// TwinCAT 3 PLC project Fraktal_Modules
// Title: Fraktal_Modules
// Company: fraktal-automation
// Author: fraktal-automation
// ProjectVersion: 0.1.0.2
// Description: Reusable Fraktal module library: cylinder CMs, clamp EM, simulation models, and configured device presets. Reason bands 10100s/11000s per Core 8.8.
// ProgramVersion: 3.1.4024.0
// libraries:
//   Tc2_Standard, * (Beckhoff Automation GmbH)
//   Tc2_System, * (Beckhoff Automation GmbH)
//   Tc2_Utilities, * (Beckhoff Automation GmbH)
//   Tc3_Module, * (Beckhoff Automation GmbH)
//   Fraktal_Core, 0.1.0.3 (fraktal-automation)
// project tree:
//   DUTs/ E_ConfigurableCylinderCommand.TcDUT, E_ClampCommand.TcDUT, E_CylinderCommand.TcDUT, E_CylinderPosition.TcDUT, E_PowerGroupCommand.TcDUT, ST_TwoHandHal.TcDUT, ST_TwoHandParCfg.TcDUT, ST_TwoHandParCmd.TcDUT, ST_TwoHandOutCmd.TcDUT, ST_TwoHandOutImm.TcDUT, ST_PneumaticPressParCfg.TcDUT, ST_PneumaticPressParCmd.TcDUT, ST_PneumaticPressOutCmd.TcDUT, ST_PneumaticPressOutImm.TcDUT, ST_PowerGroupHal.TcDUT, ST_PowerGroupParCfg.TcDUT, ST_PowerGroupParCmd.TcDUT, ST_PowerGroupOutCmd.TcDUT, ST_PowerGroupOutImm.TcDUT, ST_ConfigurableCylinderParCfg.TcDUT, ST_ConfigurableCylinderParCmd.TcDUT, ST_ConfigurableCylinderOutCmd.TcDUT, ST_ConfigurableCylinderOutImm.TcDUT, ST_ConfigurableCylinderHal.TcDUT, ST_ClampParCfg.TcDUT, ST_ClampStationParCfg.TcDUT, ST_ClampStationParCmd.TcDUT, ST_ClampStationOutCmd.TcDUT, ST_ClampStationOutImm.TcDUT, ST_ClampParCmd.TcDUT, ST_ClampOutCmd.TcDUT, ST_ClampOutImm.TcDUT, ST_CylinderHal.TcDUT, ST_CylinderParCfg.TcDUT, ST_CylinderParCmd.TcDUT, ST_CylinderOutCmd.TcDUT, ST_CylinderOutImm.TcDUT, ST_CylinderIoIdentity.TcDUT, ST_DigitalInputHal.TcDUT, ST_DigitalInputOutImm.TcDUT, ST_AirPressureHal.TcDUT, ST_AirPressureOutImm.TcDUT
//   / FB_ConfigurableCylinderCM.TcPOU, FB_ConfigurableCylinderSim.TcPOU, FB_ClampEM.TcPOU, FB_ClampStationUnit.TcPOU, FB_CylinderCM.TcPOU, FB_DigitalInputCM.TcPOU, FB_AirPressureMonitorCM.TcPOU, FB_CylinderSim.TcPOU, FB_Iv3VisionCM.TcPOU, FB_Matrix220CM.TcPOU, FB_PowerGroupCM.TcPOU, FB_TwoHandStartCM.TcPOU
//   Params/ PL_ModuleReasons.TcGVL

// ---- DUTs/E_ConfigurableCylinderCommand.TcDUT
{attribute 'qualified_only'}
TYPE E_ConfigurableCylinderCommand : (NONE := 0, TO_HOME := 1, TO_WORK := 2) DINT;
END_TYPE

// ---- DUTs/E_ClampCommand.TcDUT
{attribute 'qualified_only'}
TYPE E_ClampCommand : (NONE := 0, CLAMP := 1, UNCLAMP := 2) DINT;
END_TYPE

// ---- DUTs/E_CylinderCommand.TcDUT
{attribute 'qualified_only'}
TYPE E_CylinderCommand : (NONE := 0, EXTEND := 1, RETRACT := 2) DINT;
END_TYPE

// ---- DUTs/E_CylinderPosition.TcDUT
// Basic cylinder position (Home = retracted rest, Work = extended active).
{attribute 'qualified_only'}
TYPE E_CylinderPosition : (UNKNOWN := 0, HOME := 1, WORK := 2, MID := 3) DINT;
END_TYPE

// ---- DUTs/E_PowerGroupCommand.TcDUT
{attribute 'qualified_only'}
TYPE E_PowerGroupCommand : (NONE := 0, POWER_ON := 1, POWER_OFF := 2) DINT;
END_TYPE

// ---- DUTs/ST_TwoHandHal.TcDUT
// Raw button status plus the certified safety application's evaluated result.
// SafeActive is never calculated by the standard PLC in a real machine.
TYPE ST_TwoHandHal :
STRUCT
    LeftPressed     : BOOL;
    RightPressed    : BOOL;
    SafeActive      : BOOL;
    FieldbusHealthy : BOOL;
END_STRUCT
END_TYPE

// ---- DUTs/ST_TwoHandParCfg.TcDUT
TYPE ST_TwoHandParCfg :
STRUCT
    SchemaVersion : UINT := 1;
    RequireReleaseBetweenCycles : BOOL := TRUE;
END_STRUCT
END_TYPE

// ---- DUTs/ST_TwoHandParCmd.TcDUT
TYPE ST_TwoHandParCmd :
STRUCT
    Reserved : BOOL;
END_STRUCT
END_TYPE

// ---- DUTs/ST_TwoHandOutCmd.TcDUT
TYPE ST_TwoHandOutCmd :
STRUCT
    StartAccepted : BOOL;
END_STRUCT
END_TYPE

// ---- DUTs/ST_TwoHandOutImm.TcDUT
TYPE ST_TwoHandOutImm :
STRUCT
    LeftPressed     : BOOL;
    RightPressed    : BOOL;
    SafeActive      : BOOL;
    Armed           : BOOL;
    StartPulse      : BOOL;
    FieldbusHealthy : BOOL;
    Diagnostic      : ST_Diagnostic;
END_STRUCT
END_TYPE

// ---- DUTs/ST_PneumaticPressParCfg.TcDUT
// Core §3.8 ParCfg (SchemaVersion first; adding a member = schema change).
// v2 adds the §8.11 performance references: per-model ideal cycle (OEE
// Performance denominator, §8.5.1) and the WORK-time degradation baseline
// (§8.11.4(d); 0 = watch off).
TYPE ST_PneumaticPressParCfg :
STRUCT
    SchemaVersion       : UINT := 2;
    PressSettleTime     : TIME := T#500MS;
    TransferSettleTime  : TIME := T#100MS;
    RequireTwoHandStart : BOOL := TRUE;
    IdealCycleMs        : UDINT := 0;    // §8.5.1 — 0 = Performance not computed
    BaselineWorkMs      : UDINT := 0;    // §8.11.4(d) — 0 = degradation watch off
END_STRUCT
END_TYPE

// ---- DUTs/ST_PneumaticPressParCmd.TcDUT
TYPE ST_PneumaticPressParCmd :
STRUCT
    Reserved : BOOL;
END_STRUCT
END_TYPE

// ---- DUTs/ST_PneumaticPressOutCmd.TcDUT
TYPE ST_PneumaticPressOutCmd :
STRUCT
    CycleCompleted : BOOL;
    Homed          : BOOL;
    ChangeoverCompleted : BOOL;
END_STRUCT
END_TYPE

// ---- DUTs/ST_PneumaticPressOutImm.TcDUT
TYPE ST_PneumaticPressOutImm :
STRUCT
    PressRetracted  : BOOL;
    DoorOpen        : BOOL;
    DoorClosed      : BOOL;
    SlideInside     : BOOL;
    SlideOutside    : BOOL;
    TwoHandArmed    : BOOL;
    TwoHandActive   : BOOL;
    PartPresent     : BOOL;
    AirPressureOk   : BOOL;
    ReadyForLoad    : BOOL;
    ActiveSettleTime: TIME;
    Diagnostic      : ST_Diagnostic;
END_STRUCT
END_TYPE

// ---- DUTs/ST_PowerGroupHal.TcDUT
TYPE ST_PowerGroupHal :
STRUCT
    EnableRequestOut : BOOL; // untrusted functional request; safety system remains authoritative
    PowerFeedback    : BOOL;
    SafetyPermit     : BOOL; // read-only alias from certified safety application
    FieldbusHealthy  : BOOL;
END_STRUCT
END_TYPE

// ---- DUTs/ST_PowerGroupParCfg.TcDUT
TYPE ST_PowerGroupParCfg :
STRUCT
    SchemaVersion        : UINT := 1;
    Kind                 : E_PowerGroupKind;
    RequiredForControl   : BOOL := TRUE;
    FieldbusLossReaction : E_FieldbusLossReaction := E_FieldbusLossReaction.CONTROL_OFF;
    FeedbackTimeout      : TIME := T#2S;
END_STRUCT
END_TYPE

// ---- DUTs/ST_PowerGroupParCmd.TcDUT
TYPE ST_PowerGroupParCmd :
STRUCT
    SchemaVersion : UINT := 1;
END_STRUCT
END_TYPE

// ---- DUTs/ST_PowerGroupOutCmd.TcDUT
TYPE ST_PowerGroupOutCmd :
STRUCT
    PowerOn : BOOL;
END_STRUCT
END_TYPE

// ---- DUTs/ST_PowerGroupOutImm.TcDUT
TYPE ST_PowerGroupOutImm :
STRUCT
    Status     : ST_PowerGroupStatus;
    Diagnostic : ST_Diagnostic;
END_STRUCT
END_TYPE

// ---- DUTs/ST_ConfigurableCylinderParCfg.TcDUT
// Core §3.8 ParCfg (SchemaVersion first). Basic cylinder with optional, possibly
// REDUNDANT, position sensors. Values live in the module that needs them (§3.8a).
TYPE ST_ConfigurableCylinderParCfg :
STRUCT
    SchemaVersion     : UINT := 1;

    // --- optional & redundant sensors ---
    // count of sensors wired for each position: 0 = sensorless (time-based),
    // 1 = single, 2 = duplex (AND-combined), up to PL_Fraktal.MAX_POS_SENSORS.
    HomeSensorCount   : INT := 1;
    WorkSensorCount   : INT := 1;

    // --- timing ---
    MoveTimeout       : TIME := T#5S;    // max movement time (default 5 s)
    SettleTime        : TIME := T#30MS;  // debounce before a move is declared done
    TravelTime        : TIME := T#1S;    // sensorless travel assumption (< MoveTimeout)
    DiscrepancyTime   : TIME := T#500MS; // how long redundant sensors may disagree before fault

    // --- behaviour ---
    SingleActing      : BOOL := FALSE;   // TRUE: only ToWorkOut driven; spring return home
    SafePosOnAbort    : E_CylinderPosition := E_CylinderPosition.HOME;
    DeenergizeOnAbort : BOOL := TRUE;
END_STRUCT
END_TYPE

// ---- DUTs/ST_ConfigurableCylinderParCmd.TcDUT
TYPE ST_ConfigurableCylinderParCmd :
STRUCT
    Reserved : BOOL;
END_STRUCT
END_TYPE

// ---- DUTs/ST_ConfigurableCylinderOutCmd.TcDUT
TYPE ST_ConfigurableCylinderOutCmd :
STRUCT
    ReachedPosition : E_CylinderPosition;
END_STRUCT
END_TYPE

// ---- DUTs/ST_ConfigurableCylinderOutImm.TcDUT
TYPE ST_ConfigurableCylinderOutImm :
STRUCT
    Position   : E_CylinderPosition;
    AtHome     : BOOL;
    AtWork     : BOOL;
    Diagnostic : ST_Diagnostic;
END_STRUCT
END_TYPE

// ---- DUTs/ST_ConfigurableCylinderHal.TcDUT
// Basic cylinder HAL with REDUNDANT position sensors (safety cylinders).
// Each position has an array of sensors; only the first N (ParCfg.*SensorCount) are
// used. N = 0 -> sensorless (time-based completion). 'Arrived' = ALL present
// sensors TRUE (AND); a persistent split faults (discrepancy monitoring, §3.6.
TYPE ST_ConfigurableCylinderHal :
STRUCT
    ToWorkOut : BOOL;   // solenoid: drive to work (extend)
    ToHomeOut : BOOL;   // solenoid: drive to home (retract); single-acting leaves FALSE
    HomeFb    : ARRAY[1..PL_Fraktal.MAX_POS_SENSORS] OF BOOL;   // redundant home sensors
    WorkFb    : ARRAY[1..PL_Fraktal.MAX_POS_SENSORS] OF BOOL;   // redundant work sensors
END_STRUCT
END_TYPE

// ---- DUTs/ST_ClampParCfg.TcDUT
TYPE ST_ClampParCfg :
STRUCT
    SchemaVersion : UINT := 1;
    SettleTime    : TIME := T#150MS;
END_STRUCT
END_TYPE

// ---- DUTs/ST_ClampStationParCfg.TcDUT
TYPE ST_ClampStationParCfg :
STRUCT
    SchemaVersion : UINT := 1;
END_STRUCT
END_TYPE

// ---- DUTs/ST_ClampStationParCmd.TcDUT
TYPE ST_ClampStationParCmd :
STRUCT
    Reserved : BOOL;
END_STRUCT
END_TYPE

// ---- DUTs/ST_ClampStationOutCmd.TcDUT
TYPE ST_ClampStationOutCmd :
STRUCT
    CycleCompleted : BOOL;
END_STRUCT
END_TYPE

// ---- DUTs/ST_ClampStationOutImm.TcDUT
TYPE ST_ClampStationOutImm :
STRUCT
    Clamped   : BOOL;
    Unclamped : BOOL;
    Diagnostic: ST_Diagnostic;
END_STRUCT
END_TYPE

// ---- DUTs/ST_ClampParCmd.TcDUT
TYPE ST_ClampParCmd :
STRUCT
    Reserved : BOOL;
END_STRUCT
END_TYPE

// ---- DUTs/ST_ClampOutCmd.TcDUT
TYPE ST_ClampOutCmd :
STRUCT
    Confirmed : BOOL;
END_STRUCT
END_TYPE

// ---- DUTs/ST_ClampOutImm.TcDUT
TYPE ST_ClampOutImm :
STRUCT
    Clamped    : BOOL;
    Unclamped  : BOOL;
    Diagnostic : ST_Diagnostic;
END_STRUCT
END_TYPE

// ---- DUTs/ST_CylinderHal.TcDUT
// Annex B — cylinder HAL: 2 outputs, 2 position sensors
TYPE ST_CylinderHal :
STRUCT
    ExtendOut, RetractOut   : BOOL;
    ExtendedFb, RetractedFb : BOOL;
END_STRUCT
END_TYPE

// ---- DUTs/ST_CylinderParCfg.TcDUT
// Core §3.8: SchemaVersion FIRST, initialized to the expected version
TYPE ST_CylinderParCfg :
STRUCT
    SchemaVersion : UINT := 1;
    MoveTimeout   : TIME := T#2S;
END_STRUCT
END_TYPE

// ---- DUTs/ST_CylinderParCmd.TcDUT
TYPE ST_CylinderParCmd :
STRUCT
    Reserved : BOOL;
END_STRUCT
END_TYPE

// ---- DUTs/ST_CylinderOutCmd.TcDUT
TYPE ST_CylinderOutCmd :
STRUCT
    Reached : BOOL;
END_STRUCT
END_TYPE

// ---- DUTs/ST_CylinderOutImm.TcDUT
TYPE ST_CylinderOutImm :
STRUCT
    Extended   : BOOL;
    Retracted  : BOOL;
    ExtendedSensorTag : STRING(80);
    RetractedSensorTag: STRING(80);
    ExtendOutputTag   : STRING(80);
    RetractOutputTag  : STRING(80);
    Diagnostic : ST_Diagnostic;
END_STRUCT
END_TYPE

// ---- DUTs/ST_CylinderIoIdentity.TcDUT
// Physical identity injection for the four semantic I/O roles of a cylinder.
// The reusable CM never knows terminal models, channel numbers or project tags.
TYPE ST_CylinderIoIdentity :
STRUCT
    ExtendedSensor : ST_IoPointIdentity;
    RetractedSensor : ST_IoPointIdentity;
    ExtendOutput : ST_IoPointIdentity;
    RetractOutput : ST_IoPointIdentity;
    ExtendedTimeoutKey : STRING(255);
    RetractedTimeoutKey : STRING(255);
    BothSensorsKey : STRING(255);
END_STRUCT
END_TYPE

// ---- DUTs/ST_DigitalInputHal.TcDUT
TYPE ST_DigitalInputHal :
STRUCT
    Value : BOOL;
    Quality : BOOL := TRUE;
END_STRUCT
END_TYPE

// ---- DUTs/ST_DigitalInputOutImm.TcDUT
TYPE ST_DigitalInputOutImm :
STRUCT
    Value : BOOL;
    Quality : BOOL;
    IoTag : STRING(80);
    Diagnostic : ST_Diagnostic;
END_STRUCT
END_TYPE

// ---- DUTs/ST_AirPressureHal.TcDUT
TYPE ST_AirPressureHal :
STRUCT
    LowPressure : BOOL;
    OperatingPressure : BOOL;
    Quality : BOOL := TRUE;
END_STRUCT
END_TYPE

// ---- DUTs/ST_AirPressureOutImm.TcDUT
TYPE ST_AirPressureOutImm :
STRUCT
    LowPressure : BOOL;
    OperatingPressure : BOOL;
    PressureOk : BOOL;
    Contradictory : BOOL;
    Quality : BOOL;
    LowSensorTag : STRING(80);
    OperatingSensorTag : STRING(80);
    Diagnostic : ST_Diagnostic;
END_STRUCT
END_TYPE

// ---- Params/PL_ModuleReasons.TcGVL
{attribute 'qualified_only'}
// Core §8.8 band constants (band-extensibility rule): cylinder CM 10100-10199,
// clamp EM 11000-11999 — registered in the Core §8.8 registry.
VAR_GLOBAL CONSTANT
    CYL_NOT_EXTENDED    : DINT := 10101;
    CYL_NOT_RETRACTED   : DINT := 10102;
    CYL_BOTH_SENSORS    : DINT := 10103;
    CLAMP_NOT_CONFIRMED : DINT := 11001;
    // basic cylinder 10200-10299
    CYL_HOME_NOT_REACHED : DINT := 10111;   // timeout moving to home
    CYL_WORK_NOT_REACHED : DINT := 10112;   // timeout moving to work
    CYL_POS_IMPLAUSIBLE  : DINT := 10113;   // home AND work sensor confirmed at once (implausible)
    CYL_SENSOR_LOST      : DINT := 10114;   // confirmed position sensor dropped while holding
    CYL_DISCREPANCY      : DINT := 10116;   // redundant sensors for one position disagree > DiscrepancyTime
    CYL_CFG_INVALID      : DINT := 10115;   // TravelTime >= MoveTimeout, or no sensor+no travel
    // power-group CM 10500-10599
    POWER_ENABLE_WITHHELD : DINT := 10501;
    POWER_FEEDBACK_TIMEOUT: DINT := 10502;
    // air-pressure monitor CM 10600-10699
    AIR_SWITCH_CONFLICT    : DINT := 10601;
END_VAR

// ---- FB_ConfigurableCylinderCM.TcPOU
// Production-grade basic pneumatic cylinder Control Module (Core §2.2 base) with
// OPTIONAL and REDUNDANT position sensors (safety cylinders). Per position: 0..N
// sensors; 0 = sensorless (time-based). 'Arrived' = ALL present sensors TRUE (AND,
// safest); a persistent split of redundant sensors faults (discrepancy monitoring).
// The type is ONLY its device logic; lifecycle/timing/first-out/abort are inherited.
{attribute 'OPC.UA.DA' := '1'}
FUNCTION_BLOCK FB_ConfigurableCylinderCM EXTENDS FB_ControlModuleBase
VAR_INPUT
    Command : E_ConfigurableCylinderCommand;
    ParCfg : ST_ConfigurableCylinderParCfg;
    ParCmd : ST_ConfigurableCylinderParCmd;
END_VAR
VAR_OUTPUT
    OutCmd : ST_ConfigurableCylinderOutCmd;
    OutImm : ST_ConfigurableCylinderOutImm;
    Intlk  : FB_PermIntlk;
END_VAR
VAR
    _hal     : REFERENCE TO ST_ConfigurableCylinderHal;
    _recipe  : I_RecipeProvider;
    _tMove   : TON;
    _tSettle : TON;
    _tDiscH  : TON;                             // home discrepancy timer
    _tDiscW  : TON;                             // work discrepancy timer
    _cfgOk   : BOOL;
    _force   : BOOL;                            // SIM-only interlock force (§5.7)
    _parCfgStaged : ST_ConfigurableCylinderParCfg;
    _recipePrepared : BOOL;
END_VAR

Cyclic();

METHOD Setup : BOOL
VAR_INPUT
    Name   : STRING(80);
    HalRef : REFERENCE TO ST_ConfigurableCylinderHal;
    Recipe : I_RecipeProvider;
END_VAR
VAR
    InitialModel : ST_ModelId;
END_VAR
_M_SetName(Name);
_M_SetPresentation(DisplayNameKey := 'std.moduleType.configurableCylinder.name', DescriptionKey := 'std.moduleType.configurableCylinder.description');
_M_PublishCommand(Value := TO_DINT(E_ConfigurableCylinderCommand.TO_HOME), Label := 'std.command.toHome');   // §7.6.1 catalog
_M_PublishCommand(Value := TO_DINT(E_ConfigurableCylinderCommand.TO_WORK), Label := 'std.command.toWork');
_hal REF= HalRef;                                        // [TC3] TC3 §3.11
_recipe := Recipe;
Intlk.Define(Index := 1, Description := 'project.interlock.areaSafe', Reason := E_Reason.INTERLOCK_DROPPED, Bypassable := FALSE);
Setup := PrepareRecipe(Model := InitialModel);
IF Setup THEN CommitRecipe(); END_IF
END_METHOD

METHOD PrepareRecipe : BOOL
VAR_INPUT
    Model : ST_ModelId;
END_VAR
_parCfgStaged := ParCfg;
IF _recipe <> 0 THEN
    IF NOT _recipe.Load(ModelCode := Model.ModelCode, RecipeKey := 'ConfigurableCylinderCM', pParCfg := ADR(_parCfgStaged), Size := SIZEOF(_parCfgStaged)) THEN
        _M_Fault(E_Reason.RECIPE_INVALID, 'std.error.recipeSchemaInvalid');
        PrepareRecipe := FALSE;
        RETURN;
    END_IF
END_IF
// counts within [0..MAX]; sensorless direction needs a usable travel time
_cfgOk := (_parCfgStaged.HomeSensorCount >= 0) AND (_parCfgStaged.HomeSensorCount <= PL_Fraktal.MAX_POS_SENSORS)
      AND (_parCfgStaged.WorkSensorCount >= 0) AND (_parCfgStaged.WorkSensorCount <= PL_Fraktal.MAX_POS_SENSORS)
      AND (_parCfgStaged.TravelTime < _parCfgStaged.MoveTimeout)
      AND ((_parCfgStaged.HomeSensorCount > 0) OR (_parCfgStaged.TravelTime > T#0S))
      AND ((_parCfgStaged.WorkSensorCount > 0) OR (_parCfgStaged.TravelTime > T#0S));
IF NOT _cfgOk THEN
    _M_FaultN(PL_ModuleReasons.CYL_CFG_INVALID, 'std.error.cylinderConfigurationInvalid');
    PrepareRecipe := FALSE;
    RETURN;
END_IF
_recipePrepared := TRUE;
PrepareRecipe := TRUE;
END_METHOD

METHOD CommitRecipe
IF _recipePrepared THEN ParCfg := _parCfgStaged; END_IF
_recipePrepared := FALSE;
END_METHOD

METHOD AbortRecipe
_recipePrepared := FALSE;
END_METHOD

// TRUE iff EVERY wired sensor for the position reads TRUE (AND-combine, safest).
// Count = 0 -> not sensor-decided (caller uses the time path).
METHOD PROTECTED _M_PosArrived : BOOL
VAR_INPUT
    Work : BOOL;    // TRUE = work position, FALSE = home
END_VAR
VAR
    i, n : INT;
    all  : BOOL;
END_VAR
n := SEL(Work, ParCfg.HomeSensorCount, ParCfg.WorkSensorCount);
IF n <= 0 THEN
    _M_PosArrived := FALSE;      // no sensors: caller must use the time-based path
    RETURN;
END_IF
all := TRUE;
FOR i := 1 TO n DO
    IF Work THEN
        IF NOT _hal.WorkFb[i] THEN all := FALSE; END_IF
    ELSE
        IF NOT _hal.HomeFb[i] THEN all := FALSE; END_IF
    END_IF
END_FOR
_M_PosArrived := all;
END_METHOD

// TRUE iff the position's redundant sensors DISAGREE (at least one TRUE and at
// least one FALSE) — the discrepancy condition. Single/zero sensor => never split.
METHOD PROTECTED _M_PosSplit : BOOL
VAR_INPUT
    Work : BOOL;
END_VAR
VAR
    i, n : INT;
    anyT, anyF : BOOL;
END_VAR
n := SEL(Work, ParCfg.HomeSensorCount, ParCfg.WorkSensorCount);
IF n < 2 THEN
    _M_PosSplit := FALSE;
    RETURN;
END_IF
FOR i := 1 TO n DO
    IF Work THEN
        IF _hal.WorkFb[i] THEN anyT := TRUE; ELSE anyF := TRUE; END_IF
    ELSE
        IF _hal.HomeFb[i] THEN anyT := TRUE; ELSE anyF := TRUE; END_IF
    END_IF
END_FOR
_M_PosSplit := anyT AND anyF;
END_METHOD

// live position resolve + discrepancy monitoring (both positions, every scan)
METHOD PROTECTED OnCyclic : DINT
OnCyclic := SUPER^.OnCyclic();
Intlk.Cond[1] := NOT _force;
Intlk();
IF NOT __ISVALIDREF(_hal) THEN
    RETURN;
END_IF
OutImm.AtHome := (ParCfg.HomeSensorCount > 0) AND _M_PosArrived(Work := FALSE);
OutImm.AtWork := (ParCfg.WorkSensorCount > 0) AND _M_PosArrived(Work := TRUE);

// discrepancy monitoring — a persistent split of redundant sensors is a fault
_tDiscH(IN := _M_PosSplit(Work := FALSE), PT := ParCfg.DiscrepancyTime);
_tDiscW(IN := _M_PosSplit(Work := TRUE),  PT := ParCfg.DiscrepancyTime);
IF (_tDiscH.Q OR _tDiscW.Q) AND (_exec <> E_ExecState.ERROR) THEN
    _M_FaultN(PL_ModuleReasons.CYL_DISCREPANCY, 'std.error.cylinderSensorDiscrepancy');
END_IF

// resolve position (AtHome/AtWork already AND-combined)
IF OutImm.AtHome AND OutImm.AtWork THEN
    OutImm.Position := E_CylinderPosition.UNKNOWN;
ELSIF OutImm.AtHome THEN OutImm.Position := E_CylinderPosition.HOME;
ELSIF OutImm.AtWork THEN OutImm.Position := E_CylinderPosition.WORK;
ELSIF (ParCfg.HomeSensorCount > 0) OR (ParCfg.WorkSensorCount > 0) THEN OutImm.Position := E_CylinderPosition.MID;
END_IF
OutImm.Diagnostic := Status.Diagnostic;

// both-positions-active plausibility while idle
IF (_exec = E_ExecState.READY) AND OutImm.AtHome AND OutImm.AtWork THEN
    _M_FaultN(PL_ModuleReasons.CYL_POS_IMPLAUSIBLE, 'std.error.cylinderPositionImplausible');
END_IF
END_METHOD

// §3.14.2 — fail-safe abort
METHOD PROTECTED OnAbort : DINT
OnAbort := SUPER^.OnAbort();
IF NOT __ISVALIDREF(_hal) THEN
    RETURN;
END_IF
IF ParCfg.DeenergizeOnAbort THEN
    _hal.ToWorkOut := FALSE;
    _hal.ToHomeOut := FALSE;
ELSIF ParCfg.SafePosOnAbort = E_CylinderPosition.WORK THEN
    _hal.ToWorkOut := TRUE;  _hal.ToHomeOut := FALSE;
ELSE
    _hal.ToWorkOut := FALSE; _hal.ToHomeOut := NOT ParCfg.SingleActing;
END_IF
END_METHOD

// §5.7 SIM-only
METHOD SimForceInterlock : BOOL
VAR_INPUT
    Ok : BOOL;
END_VAR
_force := NOT Ok;
SimForceInterlock := TRUE;
END_METHOD

// drive -> await (all-sensors-agree, or time when sensorless) -> settle -> done
METHOD PROTECTED _M_Dispatch
VAR
    toWork  : BOOL;
    n       : INT;
    arrived : BOOL;
    d       : ST_Diagnostic;
END_VAR
IF _manualReq THEN
    _manualReq := FALSE;                        // §7.6.1: apply the manual command value
    Command := _manualCmd;                      // routed THROUGH dispatch — interlocks still apply
END_IF
IF (Command <> E_ConfigurableCylinderCommand.TO_HOME) AND (Command <> E_ConfigurableCylinderCommand.TO_WORK) THEN
    _M_Fault(E_Reason.UNSUPPORTED_COMMAND, 'std.error.unsupportedCylinderCommand');
    RETURN;
END_IF
IF Command = E_ConfigurableCylinderCommand.TO_WORK THEN
    _M_TagCommand(Id := 2, Label := 'std.command.toWork');
    toWork := TRUE;
ELSE
    _M_TagCommand(Id := 1, Label := 'std.command.toHome');
    toWork := FALSE;
END_IF
IF NOT Intlk.AllOk THEN
    _hal.ToWorkOut := FALSE;
    _hal.ToHomeOut := FALSE;
    d := Intlk.Diagnostic;
    d.SourcePath := _name;
    _M_FaultDiag(d);
    RETURN;
END_IF
n := SEL(toWork, ParCfg.HomeSensorCount, ParCfg.WorkSensorCount);   // sensors on the TARGET position
CASE _step OF
    10:
        OutCmd.ReachedPosition := E_CylinderPosition.UNKNOWN;
        _hal.ToWorkOut := toWork;
        _hal.ToHomeOut := (NOT toWork) AND (NOT ParCfg.SingleActing);
        _tMove(IN := FALSE);
        _tSettle(IN := FALSE);
        _step := 20;
    20:  // await arrival
        _tMove(IN := TRUE, PT := ParCfg.MoveTimeout);
        IF n > 0 THEN
            arrived := _M_PosArrived(Work := toWork);        // ALL sensors agree
        ELSE
            _tSettle(IN := TRUE, PT := ParCfg.TravelTime);      // sensorless -> travel time
            arrived := _tSettle.Q;
        END_IF
        IF arrived THEN
            _tSettle(IN := FALSE);
            _step := 30;
        ELSIF _tMove.Q THEN
            _tMove(IN := FALSE);
            _M_FaultN(SEL(toWork, PL_ModuleReasons.CYL_HOME_NOT_REACHED, PL_ModuleReasons.CYL_WORK_NOT_REACHED),
                      SEL(toWork, 'std.error.cylinderHomeTimeout', 'std.error.cylinderWorkTimeout'));
        END_IF
    30:  // settle/debounce; re-confirm all sensors still agree
        _tSettle(IN := TRUE, PT := ParCfg.SettleTime);
        IF n <= 0 THEN
            OutCmd.ReachedPosition := SEL(toWork, E_CylinderPosition.HOME, E_CylinderPosition.WORK);
            _M_Complete();
        ELSIF _M_PosArrived(Work := toWork) THEN
            IF _tSettle.Q THEN
                OutCmd.ReachedPosition := SEL(toWork, E_CylinderPosition.HOME, E_CylinderPosition.WORK);
                _M_Complete();
            END_IF
        ELSE
            _tSettle(IN := FALSE);
            _step := 20;                                     // lost agreement; keep waiting in MoveTimeout
        END_IF
ELSE
    _M_Fault(E_Reason.STEP_STALLED, 'std.error.undefinedStep');
END_CASE
END_METHOD

PROPERTY AtPos : E_CylinderPosition
GET
AtPos := OutImm.Position;
END_GET
END_PROPERTY

METHOD PROTECTED _M_PublishStatus
SUPER^._M_PublishStatus();
OutImm.Diagnostic := Status.Diagnostic;
END_METHOD

END_FUNCTION_BLOCK

// ---- FB_ConfigurableCylinderSim.TcPOU
// §5.7 sim plant for FB_ConfigurableCylinderCM with redundant sensors: after a travel time
// it sets all HomeFb[1..HomeN] / WorkFb[1..WorkN] together. StuckWork[i]/StuckHome[i]
// pin a sensor OFF so a test can inject a discrepancy.
FUNCTION_BLOCK FB_ConfigurableCylinderSim
VAR_INPUT
    Travel : TIME := T#100MS;
    HomeN  : INT := 1;
    WorkN  : INT := 1;
    StuckHome : ARRAY[1..PL_Fraktal.MAX_POS_SENSORS] OF BOOL;   // TRUE = pin this sensor OFF
    StuckWork : ARRAY[1..PL_Fraktal.MAX_POS_SENSORS] OF BOOL;
END_VAR
VAR
    _hal : REFERENCE TO ST_ConfigurableCylinderHal;
    _tW, _tH : TON;
    i : INT;
END_VAR

IF NOT __ISVALIDREF(_hal) THEN
    RETURN;
END_IF
_tW(IN := _hal.ToWorkOut, PT := Travel);
IF _tW.Q THEN
    FOR i := 1 TO WorkN DO _hal.WorkFb[i] := NOT StuckWork[i]; END_FOR
    FOR i := 1 TO HomeN DO _hal.HomeFb[i] := FALSE; END_FOR
END_IF
_tH(IN := _hal.ToHomeOut OR (NOT _hal.ToWorkOut AND NOT _hal.ToHomeOut), PT := Travel);
IF _tH.Q THEN
    FOR i := 1 TO HomeN DO _hal.HomeFb[i] := NOT StuckHome[i]; END_FOR
    FOR i := 1 TO WorkN DO _hal.WorkFb[i] := FALSE; END_FOR
END_IF

METHOD Setup : BOOL
VAR_INPUT
    HalRef : REFERENCE TO ST_ConfigurableCylinderHal;
    TravelTime : TIME;
    Home : INT;
    Work : INT;
END_VAR
VAR
    j : INT;
END_VAR
_hal REF= HalRef;
Travel := TravelTime;
HomeN := Home;
WorkN := Work;
FOR j := 1 TO HomeN DO _hal.HomeFb[j] := TRUE; END_FOR   // start at home, all agree
Setup := TRUE;
END_METHOD

END_FUNCTION_BLOCK

// ---- FB_ClampEM.TcPOU
// Annex B on the EM base: orchestration only, no device logic (§3.5); rollup §8.2.
{attribute 'OPC.UA.DA' := '1'}
FUNCTION_BLOCK FB_ClampEM EXTENDS FB_EquipmentModuleBase
VAR_INPUT
    Command : E_ClampCommand;
    ParCfg : ST_ClampParCfg;
    ParCmd : ST_ClampParCmd;
END_VAR
VAR_OUTPUT
    CylA, CylB : FB_CylinderCM;
    OutCmd : ST_ClampOutCmd;
    OutImm : ST_ClampOutImm;
END_VAR
VAR
    _recipe : I_RecipeProvider;
    _tSettle : TON;
    _parCfgStaged : ST_ClampParCfg;
    _recipePrepared : BOOL;
END_VAR

Cyclic();

METHOD PROTECTED OnCyclic : DINT
OnCyclic := SUPER^.OnCyclic();
_M_TickChildren();                       // children stay live (Annex B §B.3)
OutImm.Diagnostic := Status.Diagnostic;
END_METHOD

METHOD PrepareRecipe : BOOL
VAR_INPUT
    Model : ST_ModelId;
END_VAR
IF _recipe = 0 THEN
    _parCfgStaged := ParCfg;
    _recipePrepared := TRUE;
ELSIF _recipe.Load(ModelCode := Model.ModelCode, RecipeKey := 'ClampEM', pParCfg := ADR(_parCfgStaged), Size := SIZEOF(_parCfgStaged)) THEN
    _recipePrepared := TRUE;
ELSE
    _M_Fault(E_Reason.RECIPE_INVALID, 'std.error.recipeSchemaInvalid');
    _recipePrepared := FALSE;
    PrepareRecipe := FALSE;
    RETURN;
END_IF
PrepareRecipe := SUPER^.PrepareRecipe(Model := Model);
IF NOT PrepareRecipe THEN _recipePrepared := FALSE; END_IF
END_METHOD

METHOD CommitRecipe
SUPER^.CommitRecipe();
IF _recipePrepared THEN ParCfg := _parCfgStaged; END_IF
_recipePrepared := FALSE;
END_METHOD

METHOD AbortRecipe
SUPER^.AbortRecipe();
_recipePrepared := FALSE;
END_METHOD

METHOD Setup : BOOL
VAR_INPUT
    Name : STRING(80);
    HalA : REFERENCE TO ST_CylinderHal;
    HalB : REFERENCE TO ST_CylinderHal;
    Recipe : I_RecipeProvider;
END_VAR
VAR
    InitialModel : ST_ModelId;
END_VAR
_M_SetName(Name);
_M_SetPresentation(DisplayNameKey := 'std.moduleType.clamp.name', DescriptionKey := 'std.moduleType.clamp.description');
_recipe := Recipe;
CylA.Setup(Name := CONCAT(Name, '.CylA'), HalRef := HalA, Recipe := Recipe);
CylB.Setup(Name := CONCAT(Name, '.CylB'), HalRef := HalB, Recipe := Recipe);
_M_Register(CylA);
_M_Register(CylB);
_M_PublishCommand(Value := TO_DINT(E_ClampCommand.CLAMP), Label := 'std.command.clamp');
_M_PublishCommand(Value := TO_DINT(E_ClampCommand.UNCLAMP), Label := 'std.command.unclamp');
Setup := PrepareRecipe(Model := InitialModel);
IF Setup THEN CommitRecipe(); END_IF
END_METHOD

METHOD PROTECTED _M_Dispatch
VAR
    dir : E_CylinderCommand;
    ext : BOOL;
END_VAR
IF _manualReq THEN
    _manualReq := FALSE;
    IF (_manualCmd = TO_DINT(E_ClampCommand.CLAMP)) OR (_manualCmd = TO_DINT(E_ClampCommand.UNCLAMP)) THEN
        Command := _manualCmd;
    ELSE
        _M_Fault(E_Reason.UNSUPPORTED_COMMAND, 'std.error.unsupportedClampCommand');
        RETURN;
    END_IF
END_IF
IF (Command <> E_ClampCommand.CLAMP) AND (Command <> E_ClampCommand.UNCLAMP) THEN
    _M_Fault(E_Reason.UNSUPPORTED_COMMAND, 'std.error.unsupportedClampCommand');
    RETURN;
END_IF
ext := (Command = E_ClampCommand.CLAMP);
dir := SEL(ext, E_CylinderCommand.RETRACT, E_CylinderCommand.EXTEND);
IF ext THEN
    _M_TagCommand(Id := 1, Label := 'std.command.clamp');
ELSE
    _M_TagCommand(Id := 2, Label := 'std.command.unclamp');
END_IF
CASE _step OF
    10:  // command both cylinders in parallel (Annex B)
        OutCmd.Confirmed := FALSE;
        CylA.Abort := FALSE;
        CylB.Abort := FALSE;
        CylA.Command := dir;
        CylB.Command := dir;
        CylA.Execute := TRUE;
        CylB.Execute := TRUE;
        _tSettle(IN := FALSE);
        _step := 20;
    20:  // join on both Done — or roll up the first child Error (§8.2)
        IF CylA.Error OR CylB.Error THEN
            _M_RollupFault();
            CylA.Abort := TRUE;                    // stop the partner safely
            CylB.Abort := TRUE;
            CylA.Execute := FALSE;
            CylB.Execute := FALSE;
        ELSIF CylA.Done AND CylB.Done THEN
            CylA.Execute := FALSE;
            CylB.Execute := FALSE;
            _step := 30;
        END_IF
    30:  // settle, then confirm both feedbacks held (EM-level check, Annex B)
        _tSettle(IN := TRUE, PT := ParCfg.SettleTime);
        IF _tSettle.Q THEN
            _tSettle(IN := FALSE);
            IF (ext AND CylA.OutImm.Extended AND CylB.OutImm.Extended)
            OR ((NOT ext) AND CylA.OutImm.Retracted AND CylB.OutImm.Retracted) THEN
                OutImm.Clamped   := ext;
                OutImm.Unclamped := NOT ext;
                OutCmd.Confirmed := TRUE;
                _M_Complete();
            ELSE
                _M_FaultN(PL_ModuleReasons.CLAMP_NOT_CONFIRMED, 'project.error.clampNotConfirmedAfterSettle');
            END_IF
        END_IF
ELSE
    _M_Fault(E_Reason.STEP_STALLED, 'std.error.undefinedStep');
END_CASE
END_METHOD

METHOD PROTECTED _M_PublishStatus
SUPER^._M_PublishStatus();
OutImm.Diagnostic := Status.Diagnostic;
END_METHOD

END_FUNCTION_BLOCK

// ---- FB_CylinderCM.TcPOU
// Annex A/B pattern on the base class: the type is ONLY its device logic.
{attribute 'OPC.UA.DA' := '1'}
FUNCTION_BLOCK FB_CylinderCM EXTENDS FB_ControlModuleBase
VAR_INPUT
    Command : E_CylinderCommand;
    ParCfg : ST_CylinderParCfg;
    ParCmd : ST_CylinderParCmd;
END_VAR
VAR_OUTPUT
    OutCmd : ST_CylinderOutCmd;
    OutImm : ST_CylinderOutImm;
    Intlk  : FB_PermIntlk;
END_VAR
VAR
    _hal    : REFERENCE TO ST_CylinderHal;
    _recipe : I_RecipeProvider;
    _tMove  : TON;
    _force  : BOOL;                     // SIM hook — wrap in {IF defined (SIM_HOOKS)} for release (§5.7)
    _parCfgStaged : ST_CylinderParCfg;
    _recipePrepared : BOOL;
    _directionPermitsConfigured : BOOL;
    _extendPermit, _retractPermit : BOOL := TRUE;
    _extendPermitKey, _retractPermitKey : STRING(255);
    _extendedSensorTag, _retractedSensorTag : STRING(80);
    _extendedSensorAddress, _retractedSensorAddress : STRING(80);
    _extendOutputTag, _retractOutputTag : STRING(80);
    _extendedTimeoutKey, _retractedTimeoutKey, _bothSensorsKey : STRING(255);
    _bothSensorTags, _bothSensorAddresses : STRING(80);
END_VAR

Cyclic();

METHOD PROTECTED OnCyclic : DINT
OnCyclic := SUPER^.OnCyclic();
Intlk.Cond[1] := NOT _force;            // real application: area-safe/air-ok signals (LD/ST, §5.5)
IF NOT _directionPermitsConfigured OR (Command = E_CylinderCommand.NONE) THEN
    Intlk.Cond[2] := TRUE;
ELSIF Command = E_CylinderCommand.EXTEND THEN
    Intlk.Cond[2] := _extendPermit;
ELSIF Command = E_CylinderCommand.RETRACT THEN
    Intlk.Cond[2] := _retractPermit;
ELSE
    Intlk.Cond[2] := FALSE;
END_IF
Intlk();
IF __ISVALIDREF(_hal) THEN              // defensive (§5.6) [TC3]
    OutImm.Extended  := _hal.ExtendedFb;
    OutImm.Retracted := _hal.RetractedFb;
END_IF
OutImm.ExtendedSensorTag := _extendedSensorTag;
OutImm.RetractedSensorTag := _retractedSensorTag;
OutImm.ExtendOutputTag := _extendOutputTag;
OutImm.RetractOutputTag := _retractOutputTag;
OutImm.Diagnostic := Status.Diagnostic;
END_METHOD

// Schematic identity is application configuration, not device behavior.
// Diagnostics keep SourcePath as this module and add the exact failed channel.
METHOD ConfigureIoIdentity
VAR_INPUT
    Identity : ST_CylinderIoIdentity;
END_VAR
_extendedSensorTag := Identity.ExtendedSensor.Tag;
_extendedSensorAddress := Identity.ExtendedSensor.Address;
_retractedSensorTag := Identity.RetractedSensor.Tag;
_retractedSensorAddress := Identity.RetractedSensor.Address;
_extendOutputTag := Identity.ExtendOutput.Tag;
_retractOutputTag := Identity.RetractOutput.Tag;
_extendedTimeoutKey := Identity.ExtendedTimeoutKey;
_retractedTimeoutKey := Identity.RetractedTimeoutKey;
_bothSensorsKey := Identity.BothSensorsKey;
_bothSensorTags := CONCAT(Identity.ExtendedSensor.Tag, CONCAT(' / ', Identity.RetractedSensor.Tag));
_bothSensorAddresses := CONCAT(Identity.ExtendedSensor.Address, CONCAT(' / ', Identity.RetractedSensor.Address));
END_METHOD

// Functional stop used by an owning sequence on abort/interlock loss.
// This is not a certified stop; the safety system remains authoritative.
METHOD WithdrawOutputs
IF __ISVALIDREF(_hal) THEN
    _hal.ExtendOut := FALSE;
    _hal.RetractOut := FALSE;
END_IF
END_METHOD

METHOD PROTECTED OnAbort : DINT
OnAbort := SUPER^.OnAbort();            // base first (§3.14.2)
IF __ISVALIDREF(_hal) THEN
    _hal.ExtendOut := FALSE;
    _hal.RetractOut := FALSE;
END_IF
END_METHOD

METHOD PrepareRecipe : BOOL
VAR_INPUT
    Model : ST_ModelId;
END_VAR
IF _recipe = 0 THEN
    _parCfgStaged := ParCfg;
    _recipePrepared := TRUE;
    PrepareRecipe := TRUE;
ELSIF _recipe.Load(ModelCode := Model.ModelCode, RecipeKey := 'CylinderCM', pParCfg := ADR(_parCfgStaged), Size := SIZEOF(_parCfgStaged)) THEN
    _recipePrepared := TRUE;
    PrepareRecipe := TRUE;
ELSE
    _M_Fault(E_Reason.RECIPE_INVALID, 'std.error.recipeSchemaInvalid');
    _recipePrepared := FALSE;
    PrepareRecipe := FALSE;
END_IF
END_METHOD

METHOD CommitRecipe
IF _recipePrepared THEN ParCfg := _parCfgStaged; END_IF
_recipePrepared := FALSE;
END_METHOD

METHOD AbortRecipe
_recipePrepared := FALSE;
END_METHOD

METHOD Setup : BOOL
VAR_INPUT
    Name   : STRING(80);
    HalRef : REFERENCE TO ST_CylinderHal;
    Recipe : I_RecipeProvider;
END_VAR
VAR
    InitialModel : ST_ModelId;
END_VAR
_M_SetName(Name);
_M_SetPresentation(DisplayNameKey := 'std.moduleType.cylinder.name', DescriptionKey := 'std.moduleType.cylinder.description');
_hal REF= HalRef;                        // [TC3] TC3 §3.11
_recipe := Recipe;
Intlk.Define(Index := 1, Description := 'project.interlock.areaSafe', Reason := E_Reason.INTERLOCK_DROPPED, Bypassable := FALSE);
Intlk.Define(Index := 2, Description := 'std.interlock.directionPermitted', Reason := E_Reason.INTERLOCK_DROPPED, Bypassable := FALSE);
_M_PublishCommand(Value := TO_DINT(E_CylinderCommand.EXTEND), Label := 'std.command.extend');
_M_PublishCommand(Value := TO_DINT(E_CylinderCommand.RETRACT), Label := 'std.command.retract');
Setup := PrepareRecipe(Model := InitialModel);
IF Setup THEN CommitRecipe(); END_IF
END_METHOD

// §5.7 SIM-only force hook — wrap body in {IF defined (SIM_HOOKS)} for release builds
METHOD SimForceInterlock : BOOL
VAR_INPUT
    Id : INT;
    Ok : BOOL;
END_VAR
_force := NOT Ok;
SimForceInterlock := TRUE;
END_METHOD

METHOD PROTECTED _M_Dispatch
VAR
    ext : BOOL;
    d   : ST_Diagnostic;
END_VAR
IF _manualReq THEN
    _manualReq := FALSE;
    IF (_manualCmd = TO_DINT(E_CylinderCommand.EXTEND)) OR (_manualCmd = TO_DINT(E_CylinderCommand.RETRACT)) THEN
        Command := _manualCmd;
    ELSE
        _M_Fault(E_Reason.UNSUPPORTED_COMMAND, 'std.error.unsupportedCylinderCommand');
        RETURN;
    END_IF
END_IF
IF (Command <> E_CylinderCommand.EXTEND) AND (Command <> E_CylinderCommand.RETRACT) THEN
    _M_Fault(E_Reason.UNSUPPORTED_COMMAND, 'std.error.unsupportedCylinderCommand');
    RETURN;
END_IF
IF Command = E_CylinderCommand.EXTEND THEN
    _M_TagCommand(Id := 1, Label := 'std.command.extend');       // §8.11.4(a)
    IF _directionPermitsConfigured THEN
        Intlk.Define(Index := 2, Description := _extendPermitKey, Reason := E_Reason.INTERLOCK_DROPPED, Bypassable := FALSE);
        Intlk.Cond[2] := _extendPermit;
    ELSE
        Intlk.Cond[2] := TRUE;
    END_IF
ELSE
    _M_TagCommand(Id := 2, Label := 'std.command.retract');
    IF _directionPermitsConfigured THEN
        Intlk.Define(Index := 2, Description := _retractPermitKey, Reason := E_Reason.INTERLOCK_DROPPED, Bypassable := FALSE);
        Intlk.Cond[2] := _retractPermit;
    ELSE
        Intlk.Cond[2] := TRUE;
    END_IF
END_IF
Intlk();
IF NOT Intlk.AllOk THEN
    _hal.ExtendOut := FALSE;
    _hal.RetractOut := FALSE;
    d := Intlk.Diagnostic;
    d.SourcePath := _name;                            // owner sets the path (§7.2)
    _M_FaultDiag(d);
    RETURN;
END_IF
IF _hal.ExtendedFb AND _hal.RetractedFb THEN
    IF _bothSensorsKey <> '' THEN
        _M_FaultIoN(Code := PL_ModuleReasons.CYL_BOTH_SENSORS, Text := _bothSensorsKey,
            IoTag := _bothSensorTags, IoAddress := _bothSensorAddresses);
    ELSE
        _M_FaultN(Code := PL_ModuleReasons.CYL_BOTH_SENSORS, Text := 'std.error.cylinderBothSensors');
    END_IF
    RETURN;
END_IF
ext := (Command = E_CylinderCommand.EXTEND);
CASE _step OF
    10:
        OutCmd.Reached := FALSE;
        _hal.ExtendOut  := ext;
        _hal.RetractOut := NOT ext;
        _tMove(IN := FALSE);
        _step := 20;
    20:
        _tMove(IN := TRUE, PT := ParCfg.MoveTimeout);
        IF (ext AND _hal.ExtendedFb) OR ((NOT ext) AND _hal.RetractedFb) THEN
            _tMove(IN := FALSE);
            OutCmd.Reached := TRUE;
            _M_Complete();
        ELSIF _tMove.Q THEN
            _tMove(IN := FALSE);
            IF ext AND (_extendedSensorTag <> '') THEN
                _M_FaultIoN(Code := PL_ModuleReasons.CYL_NOT_EXTENDED, Text := _extendedTimeoutKey,
                    IoTag := _extendedSensorTag, IoAddress := _extendedSensorAddress);
            ELSIF (NOT ext) AND (_retractedSensorTag <> '') THEN
                _M_FaultIoN(Code := PL_ModuleReasons.CYL_NOT_RETRACTED, Text := _retractedTimeoutKey,
                    IoTag := _retractedSensorTag, IoAddress := _retractedSensorAddress);
            ELSIF ext THEN
                _M_FaultN(Code := PL_ModuleReasons.CYL_NOT_EXTENDED, Text := 'std.error.cylinderExtendTimeout');
            ELSE
                _M_FaultN(Code := PL_ModuleReasons.CYL_NOT_RETRACTED, Text := 'std.error.cylinderRetractTimeout');
            END_IF
        END_IF
ELSE
    _M_Fault(E_Reason.STEP_STALLED, 'std.error.undefinedStep');    // defined ELSE (§5.6)
END_CASE
END_METHOD

// Functional collision/process interlocks supplied by the owning EM/Unit.
// Methods are not OPC UA writes; the check is repeated inside dispatch so manual
// commands use the same rule. Certified safety remains external.
METHOD SetDirectionalPermits
VAR_INPUT
    ExtendOk : BOOL;
    RetractOk : BOOL;
    ExtendDescriptionKey : STRING(255);
    RetractDescriptionKey : STRING(255);
END_VAR
_directionPermitsConfigured := TRUE;
_extendPermit := ExtendOk;
_retractPermit := RetractOk;
_extendPermitKey := ExtendDescriptionKey;
_retractPermitKey := RetractDescriptionKey;
END_METHOD

// Pure release-query companion to SetDirectionalPermits. The owning Unit uses
// this for act-or-explain so the HMI checks the exact permit used by dispatch.
METHOD AppendDirectionalRelease : INT
VAR_INPUT
    Value : DINT;
END_VAR
VAR_IN_OUT
    Report : ST_ReleaseReport;
END_VAR
VAR
    permitted : BOOL;
    validCommand : BOOL;
    descriptionKey : STRING(255);
END_VAR
permitted := TRUE;
validCommand := (Value = TO_DINT(E_CylinderCommand.EXTEND))
    OR (Value = TO_DINT(E_CylinderCommand.RETRACT));
descriptionKey := '';
IF _directionPermitsConfigured AND (Value = TO_DINT(E_CylinderCommand.EXTEND)) THEN
    permitted := _extendPermit;
    descriptionKey := _extendPermitKey;
ELSIF _directionPermitsConfigured AND (Value = TO_DINT(E_CylinderCommand.RETRACT)) THEN
    permitted := _retractPermit;
    descriptionKey := _retractPermitKey;
ELSIF NOT validCommand THEN
    permitted := FALSE;
    descriptionKey := 'std.error.unsupportedCylinderCommand';
ELSE
    permitted := TRUE;
END_IF
IF NOT permitted AND (Report.Count < PL_Fraktal.MAX_RELEASE_REASONS) THEN
    Report.Count := Report.Count + 1;
    Report.Reasons[Report.Count].Description := descriptionKey;
    Report.Reasons[Report.Count].SourcePath := _name;
    IF validCommand THEN
        Report.Reasons[Report.Count].ReasonCode := E_Reason.INTERLOCK_DROPPED;
    ELSE
        Report.Reasons[Report.Count].ReasonCode := E_Reason.UNSUPPORTED_COMMAND;
    END_IF
    Report.Reasons[Report.Count].Kind := E_ReleaseKind.INTERLOCK;
    Report.Reasons[Report.Count].Bypassable := FALSE;
END_IF
AppendDirectionalRelease := Report.Count;
END_METHOD

METHOD PROTECTED _M_PublishStatus
SUPER^._M_PublishStatus();
OutImm.Diagnostic := Status.Diagnostic;
END_METHOD

END_FUNCTION_BLOCK

// ---- FB_ClampStationUnit.TcPOU
// Executable root Unit: continuous Clamp -> Unclamp cycle over one Clamp EM.
{attribute 'OPC.UA.DA' := '1'}
FUNCTION_BLOCK FB_ClampStationUnit EXTENDS FB_UnitBase
VAR_INPUT
    ParCfg : ST_ClampStationParCfg;
    ParCmd : ST_ClampStationParCmd;
END_VAR
VAR_OUTPUT
    Clamp  : FB_ClampEM;
    OutCmd : ST_ClampStationOutCmd;
    OutImm : ST_ClampStationOutImm;
END_VAR

Cyclic();

METHOD Setup : BOOL
VAR_INPUT
    Name : STRING(80);
    HalA : REFERENCE TO ST_CylinderHal;
    HalB : REFERENCE TO ST_CylinderHal;
    Recipe : I_RecipeProvider;
END_VAR
_M_SetName(Name);
_M_SetPresentation(DisplayNameKey := 'project.module.clampStation.name', DescriptionKey := 'project.module.clampStation.description');
Setup := Clamp.Setup(Name := CONCAT(Name, '.Clamp'), HalA := HalA, HalB := HalB, Recipe := Recipe);
IF Setup THEN Setup := _M_Register(Clamp); END_IF
END_METHOD

METHOD PROTECTED OnCyclic : DINT
OnCyclic := SUPER^.OnCyclic();
OutImm.Clamped := Clamp.OutImm.Clamped;
OutImm.Unclamped := Clamp.OutImm.Unclamped;
END_METHOD

METHOD PROTECTED _M_Dispatch
CASE _step OF
    10:
        OutCmd.CycleCompleted := FALSE;
        _M_SetStep(StepNo := 100, StepName := 'project.step.commandClamp', Awaits := 0,
            AwaitingLabel := '', Class := E_TimeClass.WORK, ExpectedTime := T#0S);
        Clamp.Abort := FALSE;
        Clamp.Command := E_ClampCommand.CLAMP;
        Clamp.Execute := TRUE;
        _step := 20;
    20:
        _M_SetStep(StepNo := 110, StepName := 'project.step.awaitClamp', Awaits := Clamp,
            AwaitingLabel := 'Clamp.CLAMP', Class := E_TimeClass.WORK, ExpectedTime := T#0S);
        IF Clamp.Done THEN
            Clamp.Execute := FALSE;
            _step := 30;
        END_IF
    30:
        _M_SetStep(StepNo := 200, StepName := 'project.step.commandUnclamp', Awaits := 0,
            AwaitingLabel := '', Class := E_TimeClass.WORK, ExpectedTime := T#0S);
        Clamp.Abort := FALSE;
        Clamp.Command := E_ClampCommand.UNCLAMP;
        Clamp.Execute := TRUE;
        _step := 40;
    40:
        _M_SetStep(StepNo := 210, StepName := 'project.step.awaitUnclamp', Awaits := Clamp,
            AwaitingLabel := 'Clamp.UNCLAMP', Class := E_TimeClass.WORK, ExpectedTime := T#0S);
        IF Clamp.Done THEN
            Clamp.Execute := FALSE;
            _step := 50;
        END_IF
    50:
        OutCmd.CycleCompleted := TRUE;
        IF _M_EndOfCycle() THEN _step := 10; END_IF
ELSE
    _M_Fault(E_Reason.STEP_STALLED, 'std.error.undefinedStep');
END_CASE
END_METHOD

METHOD PROTECTED _M_RouteManual : BOOL
VAR_INPUT
    TargetPath : STRING(255);
    Value : DINT;
END_VAR
_M_RouteManual := FALSE;
IF TargetPath = Clamp.Name THEN
    _M_RouteManual := Clamp.ManualCommand(Value := Value);
END_IF
END_METHOD

METHOD PROTECTED _M_PublishStatus
SUPER^._M_PublishStatus();
OutImm.Diagnostic := Status.Diagnostic;
END_METHOD

END_FUNCTION_BLOCK

// ---- FB_DigitalInputCM.TcPOU
// Basic passive digital-input CM. Owning logic consumes semantic Value; the
// project catalog injects the physical identity separately from the HAL.
{attribute 'OPC.UA.DA' := '1'}
FUNCTION_BLOCK FB_DigitalInputCM EXTENDS FB_ControlModuleBase
VAR_OUTPUT
    OutImm : ST_DigitalInputOutImm;
END_VAR
VAR
    _hal : REFERENCE TO ST_DigitalInputHal;
    _identity : ST_IoPointIdentity;
END_VAR

Cyclic();

METHOD Setup : BOOL
VAR_INPUT
    Name : STRING(80);
    HalRef : REFERENCE TO ST_DigitalInputHal;
    DisplayNameKey : STRING(160);
    DescriptionKey : STRING(160);
END_VAR
_M_SetName(Name);
_M_SetPresentation(DisplayNameKey := DisplayNameKey, DescriptionKey := DescriptionKey);
_hal REF= HalRef;
Setup := __ISVALIDREF(_hal);
END_METHOD

METHOD ConfigureIoIdentity
VAR_INPUT
    Identity : ST_IoPointIdentity;
END_VAR
_identity := Identity;
END_METHOD

METHOD PROTECTED OnCyclic : DINT
OnCyclic := SUPER^.OnCyclic();
IF __ISVALIDREF(_hal) THEN
    OutImm.Value := _hal.Value;
    OutImm.Quality := _hal.Quality;
ELSE
    OutImm.Value := FALSE;
    OutImm.Quality := FALSE;
END_IF
OutImm.IoTag := _identity.Tag;
OutImm.Diagnostic := Status.Diagnostic;
END_METHOD

METHOD PROTECTED _M_Dispatch
_M_Fault(E_Reason.UNSUPPORTED_COMMAND,
    'std.error.passiveInputHasNoCommand');
END_METHOD

METHOD PROTECTED _M_PublishStatus
SUPER^._M_PublishStatus();
OutImm.Diagnostic := Status.Diagnostic;
END_METHOD

END_FUNCTION_BLOCK

// ---- FB_AirPressureMonitorCM.TcPOU
// Basic passive two-threshold pneumatic-pressure CM. Both switches active is
// implausible and faults with both exact tags; neither/high-only are status states.
{attribute 'OPC.UA.DA' := '1'}
FUNCTION_BLOCK FB_AirPressureMonitorCM EXTENDS FB_ControlModuleBase
VAR_OUTPUT
    OutImm : ST_AirPressureOutImm;
END_VAR
VAR
    _hal : REFERENCE TO ST_AirPressureHal;
    _lowIdentity, _operatingIdentity : ST_IoPointIdentity;
    _bothTags, _bothAddresses : STRING(80);
END_VAR

Cyclic();

METHOD Setup : BOOL
VAR_INPUT
    Name : STRING(80);
    HalRef : REFERENCE TO ST_AirPressureHal;
END_VAR
_M_SetName(Name);
_M_SetPresentation(DisplayNameKey := 'std.moduleType.airPressure.name',
    DescriptionKey := 'std.moduleType.airPressure.description');
_hal REF= HalRef;
Setup := __ISVALIDREF(_hal);
END_METHOD

METHOD ConfigureIoIdentity
VAR_INPUT
    LowSensor : ST_IoPointIdentity;
    OperatingSensor : ST_IoPointIdentity;
END_VAR
_lowIdentity := LowSensor;
_operatingIdentity := OperatingSensor;
_bothTags := CONCAT(LowSensor.Tag, CONCAT(' / ', OperatingSensor.Tag));
_bothAddresses := CONCAT(LowSensor.Address, CONCAT(' / ', OperatingSensor.Address));
END_METHOD

METHOD PROTECTED OnCyclic : DINT
OnCyclic := SUPER^.OnCyclic();
IF __ISVALIDREF(_hal) THEN
    OutImm.LowPressure := _hal.LowPressure;
    OutImm.OperatingPressure := _hal.OperatingPressure;
    OutImm.Quality := _hal.Quality;
    OutImm.Contradictory := _hal.LowPressure AND _hal.OperatingPressure;
    OutImm.PressureOk := _hal.OperatingPressure AND NOT _hal.LowPressure AND _hal.Quality;
    IF OutImm.Contradictory THEN
        _M_FaultIoN(Code := PL_ModuleReasons.AIR_SWITCH_CONFLICT,
            Text := 'std.error.airPressureSwitchConflict',
            IoTag := _bothTags, IoAddress := _bothAddresses);
    ELSE
        ;
    END_IF
ELSE
    OutImm.LowPressure := FALSE;
    OutImm.OperatingPressure := FALSE;
    OutImm.Quality := FALSE;
    OutImm.Contradictory := FALSE;
    OutImm.PressureOk := FALSE;
END_IF
OutImm.LowSensorTag := _lowIdentity.Tag;
OutImm.OperatingSensorTag := _operatingIdentity.Tag;
OutImm.Diagnostic := Status.Diagnostic;
END_METHOD

METHOD PROTECTED _M_Dispatch
_M_Fault(E_Reason.UNSUPPORTED_COMMAND,
    'std.error.passiveInputHasNoCommand');
END_METHOD

METHOD PROTECTED _M_PublishStatus
SUPER^._M_PublishStatus();
OutImm.Diagnostic := Status.Diagnostic;
END_METHOD

END_FUNCTION_BLOCK

// ---- FB_CylinderSim.TcPOU
// §5.7 per-type sim plant model: drives the HAL feedback with a travel time —
// shared by TcUnit suites and virtual commissioning (§2.6).
FUNCTION_BLOCK FB_CylinderSim
VAR
    Travel : TIME := T#0S;
END_VAR
VAR
    _hal : REFERENCE TO ST_CylinderHal;
    _tE, _tR : TON;
END_VAR

IF NOT __ISVALIDREF(_hal) THEN
    RETURN;
END_IF
_tE(IN := _hal.ExtendOut AND NOT _hal.ExtendedFb, PT := Travel);
IF _tE.Q THEN
    _hal.ExtendedFb  := TRUE;
    _hal.RetractedFb := FALSE;
END_IF
_tR(IN := _hal.RetractOut AND NOT _hal.RetractedFb, PT := Travel);
IF _tR.Q THEN
    _hal.RetractedFb := TRUE;
    _hal.ExtendedFb  := FALSE;
END_IF

METHOD Setup : BOOL
VAR_INPUT
    HalRef : REFERENCE TO ST_CylinderHal;
    TravelTime : TIME;
END_VAR
_hal REF= HalRef;
Travel := TravelTime;
Setup := TRUE;
END_METHOD

END_FUNCTION_BLOCK

// ---- FB_Iv3VisionCM.TcPOU
// MODEL PRESET (Core §3.15.1a): Keyence IV3 = the generic FB_TcpVisionCM with
// preconfigured protocol strings. Everything below is configuration, not code —
// a deployment could equally instantiate FB_TcpVisionCM and set these via §3.8.
// Extend further ONLY for genuinely IV3-specific features (override _M_OnResponse
// for special result formats, add commands to the §7.6.1 catalog, etc.).
// Strings are TYPICAL of the IV3 non-procedural protocol — VERIFY vs the IV3
// communication manual for the deployed model/firmware.
FUNCTION_BLOCK FB_Iv3VisionCM EXTENDS FB_TcpVisionCM
VAR
END_VAR

Cyclic();

METHOD Setup : BOOL
VAR_INPUT
    Name : STRING(80);
    Chan : I_ByteChannel;
    DevHost : STRING(80);
    DevPort : UINT;
END_VAR
ParCfg.TriggerCmd := 'T1'; // IV3 preset — VERIFY vs manual
ParCfg.OkPrefix := 'OK';
ParCfg.NgPrefix := 'NG';
Setup := SUPER^.Setup(Name := Name, Chan := Chan, DevHost := DevHost, DevPort := DevPort);
END_METHOD

END_FUNCTION_BLOCK

// ---- FB_Matrix220CM.TcPOU
// MODEL PRESET (Core §3.15.1a): Datalogic Matrix 220 = the generic
// FB_TcpCodeReaderCM with preconfigured host-mode strings. Configuration, not
// code. Extend ONLY for Matrix-specific features. VERIFY strings vs the Matrix
// host-mode manual for the deployed configuration.
FUNCTION_BLOCK FB_Matrix220CM EXTENDS FB_TcpCodeReaderCM
VAR
END_VAR

Cyclic();

METHOD Setup : BOOL
VAR_INPUT
    Name : STRING(80);
    Chan : I_ByteChannel;
    DevHost : STRING(80);
    DevPort : UINT;
END_VAR
ParCfg.TriggerCmd := 'T';  // Matrix host-mode preset — VERIFY vs manual
ParCfg.NoReadText := 'NOREAD';
Setup := SUPER^.Setup(Name := Name, Chan := Chan, DevHost := DevHost, DevPort := DevPort);
END_METHOD

END_FUNCTION_BLOCK

// ---- FB_PowerGroupCM.TcPOU
// §9.8 basic power-group CM. It requests functional enable; certified safety
// logic and field-output watchdogs remain authoritative. Recovery never self-energizes.
{attribute 'OPC.UA.DA' := '1'}
FUNCTION_BLOCK FB_PowerGroupCM EXTENDS FB_ControlModuleBase
VAR_INPUT
    Command : E_PowerGroupCommand;
    ParCfg  : ST_PowerGroupParCfg;
    ParCmd  : ST_PowerGroupParCmd;
END_VAR
VAR_OUTPUT
    OutCmd : ST_PowerGroupOutCmd;
    OutImm : ST_PowerGroupOutImm;
END_VAR
VAR
    _hal : REFERENCE TO ST_PowerGroupHal;
    _tFeedback : TON;
    _rearmRequired : BOOL;
END_VAR

Cyclic();

METHOD Setup : BOOL
VAR_INPUT
    Name : STRING(80);
    HalRef : REFERENCE TO ST_PowerGroupHal;
END_VAR
_M_SetName(Name);
_M_SetPresentation(DisplayNameKey := 'std.moduleType.powerGroup.name', DescriptionKey := 'std.moduleType.powerGroup.description');
_hal REF= HalRef;
// Power control deliberately has no MANUAL command catalog: it uses the Unit's
// POWER_CONTROL-gated ReqControlOn/ReqControlOff endpoint (§9.8).
Setup := TRUE;
END_METHOD

METHOD PROTECTED OnCyclic : DINT
VAR
    busMustDrop : BOOL;
END_VAR
OnCyclic := SUPER^.OnCyclic();
CASE ParCfg.FieldbusLossReaction OF
    E_FieldbusLossReaction.ALARM_ONLY, E_FieldbusLossReaction.STOP_UNIT:
        busMustDrop := FALSE;
    E_FieldbusLossReaction.POWER_GROUP_OFF, E_FieldbusLossReaction.CONTROL_OFF:
        busMustDrop := TRUE;
ELSE
    busMustDrop := TRUE; // unknown policy fails toward power removal
END_CASE
IF (NOT _hal.SafetyPermit) OR (busMustDrop AND NOT _hal.FieldbusHealthy) THEN
    IF _hal.EnableRequestOut OR _hal.PowerFeedback THEN _rearmRequired := TRUE; END_IF
    _hal.EnableRequestOut := FALSE;
END_IF
OutCmd.PowerOn := _hal.PowerFeedback;
OutImm.Status.Present := TRUE;
OutImm.Status.Name := _name;
OutImm.Status.Kind := ParCfg.Kind;
OutImm.Status.RequiredForControl := ParCfg.RequiredForControl;
OutImm.Status.RequestedOn := _hal.EnableRequestOut;
OutImm.Status.PowerOn := _hal.PowerFeedback;
OutImm.Status.SafetyPermit := _hal.SafetyPermit;
OutImm.Status.FieldbusHealthy := _hal.FieldbusHealthy;
OutImm.Status.FieldbusLossReaction := ParCfg.FieldbusLossReaction;
OutImm.Status.RearmRequired := _rearmRequired;
IF _hal.PowerFeedback THEN
    OutImm.Status.State := E_PowerState.ON;
ELSIF _rearmRequired THEN
    OutImm.Status.State := E_PowerState.TRIPPED;
ELSE
    OutImm.Status.State := E_PowerState.OFF;
END_IF
OutImm.Status.Diagnostic := Status.Diagnostic;
OutImm.Diagnostic := Status.Diagnostic;
ControlPower.Present := TRUE;
ControlPower.GroupCount := 1;
ControlPower.Groups[1] := OutImm.Status;
ControlPower.RequestedOn := _hal.EnableRequestOut;
ControlPower.ControlOn := _hal.PowerFeedback;
ControlPower.RearmRequired := _rearmRequired;
END_METHOD

METHOD PROTECTED _M_Dispatch
IF _manualReq THEN
    Command := _manualCmd;
    _manualReq := FALSE;
END_IF
CASE _step OF
    10:
        CASE Command OF
            E_PowerGroupCommand.POWER_ON:
                IF (NOT _hal.SafetyPermit) OR (NOT _hal.FieldbusHealthy) THEN
                    _M_FaultN(Code := PL_ModuleReasons.POWER_ENABLE_WITHHELD, Text := 'std.error.powerEnableWithheld');
                ELSE
                    _rearmRequired := FALSE;
                    _hal.EnableRequestOut := TRUE;
                    _step := 20;
                END_IF
            E_PowerGroupCommand.POWER_OFF:
                _hal.EnableRequestOut := FALSE;
                _step := 30;
        ELSE
            _M_Fault(E_Reason.UNSUPPORTED_COMMAND, 'std.error.unsupportedPowerCommand');
        END_CASE
    20:
        _tFeedback(IN := NOT _hal.PowerFeedback, PT := ParCfg.FeedbackTimeout);
        IF _hal.PowerFeedback THEN _tFeedback(IN := FALSE); _M_Complete();
        ELSIF _tFeedback.Q THEN _M_FaultN(Code := PL_ModuleReasons.POWER_FEEDBACK_TIMEOUT, Text := 'std.error.powerOnFeedbackTimeout'); END_IF
    30:
        _tFeedback(IN := _hal.PowerFeedback, PT := ParCfg.FeedbackTimeout);
        IF NOT _hal.PowerFeedback THEN _tFeedback(IN := FALSE); _M_Complete();
        ELSIF _tFeedback.Q THEN _M_FaultN(Code := PL_ModuleReasons.POWER_FEEDBACK_TIMEOUT, Text := 'std.error.powerOffFeedbackTimeout'); END_IF
ELSE
    _hal.EnableRequestOut := FALSE;
    _M_Fault(E_Reason.STEP_STALLED, 'std.error.undefinedPowerStep');
END_CASE
END_METHOD

METHOD PROTECTED OnAbort : DINT
OnAbort := SUPER^.OnAbort();
_hal.EnableRequestOut := FALSE;
_rearmRequired := TRUE;
END_METHOD

END_FUNCTION_BLOCK

// ---- FB_TwoHandStartCM.TcPOU
// Functional cycle-start edge from a certified two-hand-control result.
// This CM does not implement simultaneity, anti-tie-down, PL or safe outputs.
{attribute 'OPC.UA.DA' := '1'}
FUNCTION_BLOCK FB_TwoHandStartCM EXTENDS FB_ControlModuleBase
VAR_INPUT
    ParCfg : ST_TwoHandParCfg;
    ParCmd : ST_TwoHandParCmd;
END_VAR
VAR_OUTPUT
    OutCmd : ST_TwoHandOutCmd;
    OutImm : ST_TwoHandOutImm;
END_VAR
VAR
    _hal : REFERENCE TO ST_TwoHandHal;
    _safeRise : R_TRIG;
    _armed : BOOL;
END_VAR

Cyclic();

METHOD Setup : BOOL
VAR_INPUT
    Name : STRING(80);
    HalRef : REFERENCE TO ST_TwoHandHal;
END_VAR
_M_SetName(Name);
_M_SetPresentation(DisplayNameKey := 'std.moduleType.twoHand.name', DescriptionKey := 'std.moduleType.twoHand.description');
_hal REF= HalRef;
Setup := TRUE;
END_METHOD

METHOD PROTECTED OnCyclic : DINT
OnCyclic := SUPER^.OnCyclic();
OutImm.StartPulse := FALSE;
OutCmd.StartAccepted := FALSE;
IF __ISVALIDREF(_hal) THEN
    OutImm.LeftPressed := _hal.LeftPressed;
    OutImm.RightPressed := _hal.RightPressed;
    OutImm.FieldbusHealthy := _hal.FieldbusHealthy;
    OutImm.SafeActive := _hal.SafeActive AND _hal.FieldbusHealthy;
    IF NOT _hal.FieldbusHealthy THEN
        _armed := FALSE;
    ELSIF NOT _hal.LeftPressed AND NOT _hal.RightPressed AND NOT _hal.SafeActive THEN
        _armed := TRUE;
    END_IF
    _safeRise(CLK := OutImm.SafeActive);
    IF _safeRise.Q AND (_armed OR NOT ParCfg.RequireReleaseBetweenCycles) THEN
        OutImm.StartPulse := TRUE;
        OutCmd.StartAccepted := TRUE;
        _armed := FALSE;
    END_IF
ELSE
    OutImm.LeftPressed := FALSE;
    OutImm.RightPressed := FALSE;
    OutImm.SafeActive := FALSE;
    OutImm.FieldbusHealthy := FALSE;
    _armed := FALSE;
    _safeRise(CLK := FALSE);
END_IF
OutImm.Armed := _armed;
OutImm.Diagnostic := Status.Diagnostic;
Safety.Present := TRUE;
Safety.AllSafe := OutImm.FieldbusHealthy;
Safety.DemandActive := OutImm.LeftPressed OR OutImm.RightPressed;
Safety.FaultActive := NOT OutImm.FieldbusHealthy;
Safety.DeviceCount := 1;
Safety.Devices[1].Present := TRUE;
Safety.Devices[1].Name := _name;
Safety.Devices[1].Kind := E_SafetyDeviceKind.TWO_HAND_CONTROL;
Safety.Devices[1].Ready := OutImm.Armed;
Safety.Devices[1].DemandActive := OutImm.LeftPressed OR OutImm.RightPressed;
Safety.Devices[1].SafeStateActive := NOT OutImm.SafeActive;
Safety.Devices[1].FieldbusHealthy := OutImm.FieldbusHealthy;
Safety.Devices[1].Description := 'project.safety.twoHandControl';
END_METHOD

METHOD PROTECTED _M_Dispatch
_M_Fault(E_Reason.UNSUPPORTED_COMMAND, 'std.error.twoHandHasNoCommand');
END_METHOD

METHOD PROTECTED _M_PublishStatus
SUPER^._M_PublishStatus();
OutImm.Diagnostic := Status.Diagnostic;
END_METHOD

END_FUNCTION_BLOCK
